(* CODESYS project Johnson,Joachim,Uppgift18_V3.project

Project tree, tasks and I/O mapping:
  Device : CODESYS Control Win V3, 3S - Smart Software Solutions GmbH, order no. 305021, version 3.5.10.40
    application Application
      libraries: Standard, * (System)
      task MainTask (cyclic, interval t#20ms, priority 1) calls PLC_PRG
      program PLC_PRG [LD]
      Symbols
      global variables GVL
*)

// Device/Application/GVL
{attribute 'qualified_only'}
VAR_GLOBAL
		// signals from buttons
	iSUB00_S1: BOOL; // StartButton
	iSUB00_S2: BOOL; // Stopbutton
	iSUB00_S3: BOOL; // Resetbutton
	
	running: BOOL; // Is the aplication running
	alarm: BOOL; // Is the aplication running
	
	// Signals from conveyors
	iSUB01_B1: BOOL; // Signals för conveyor 1. ontop
	iSUB02_B1: BOOL; // Signals för conveyor 2. ontop
	iSUB03_B1: BOOL; // Signals för conveyor 3. ontop
	
	// conveyor signal ontop conveyro.
	oSUB00_H1: BOOL; // Auto-On light
	oSUB00_H2: BOOL; // Alarm light
	oSUB00_H3: WORD;
	oSUB01_K1: BOOL; // MOTOR FÖR converoyr 1
	oSUB02_K1: BOOL; // MOTOR FÖR converoyr 2
	oSUB03_K1: BOOL; // MOTOR FÖR converoyr 3
END_VAR

// Device/Application/PLC_PRG
PROGRAM PLC_PRG
VAR
	ReturnRunnongBool: BOOL;
	PressBtnTime: TIME;
	PressBtnTimer: TON;
	ONTOPCONRETURN: BOOL;
	ONTOPCONRETURN2: BOOL; // check that the previous con not take controll over engine/converour
	ONTOPCONRETURN3: BOOL; // check that the previous con not take controll over engine/converour
	PallCounter: CTU;
END_VAR
VAR // added by the converter: edge detectors and wires of the graphical bodies
    _w1, _w2, _w3, _w4 : BOOL;
END_VAR

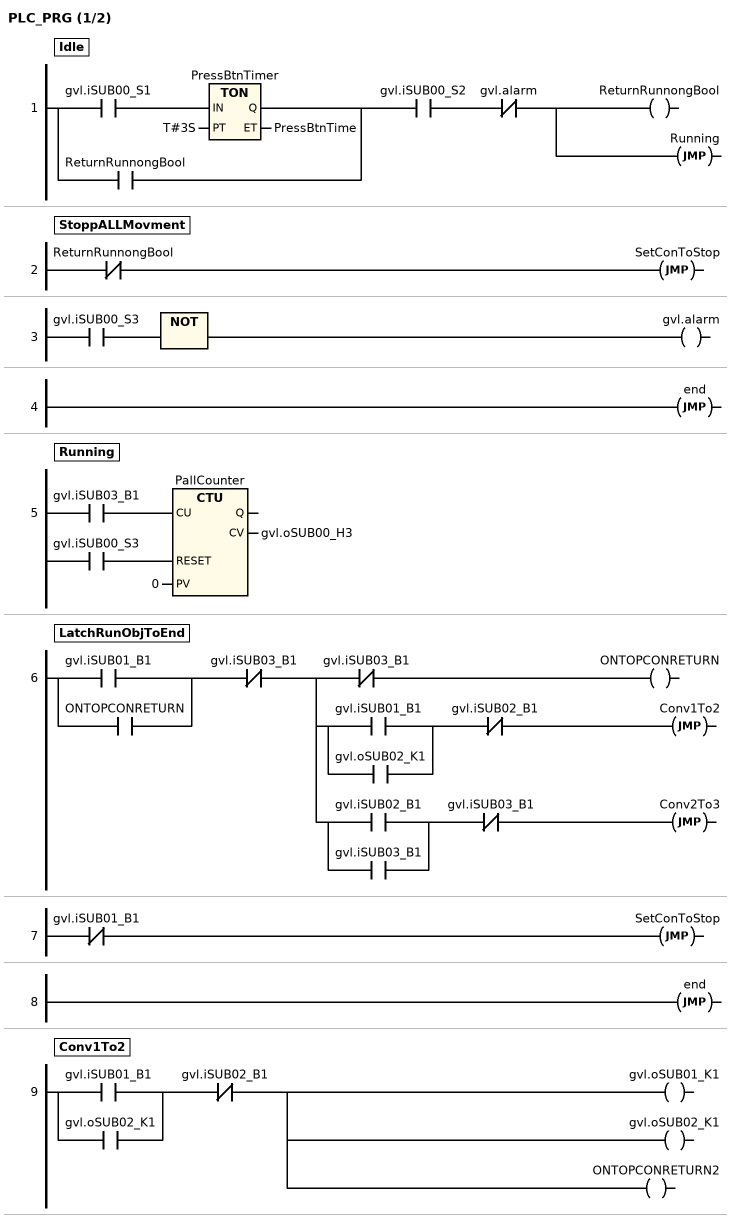
// NETWORK 1
Idle:
PressBtnTimer(IN := gvl.iSUB00_S1, PT := T#3S, ET => PressBtnTime); // TON
_w1 := (PressBtnTimer.Q OR ReturnRunnongBool) AND gvl.iSUB00_S2 AND NOT gvl.alarm;
ReturnRunnongBool := _w1;
IF _w1 THEN JMP Running; END_IF

// NETWORK 2
StoppALLMovment:
IF NOT ReturnRunnongBool THEN JMP SetConToStop; END_IF

// NETWORK 3
gvl.alarm := NOT gvl.iSUB00_S3;

// NETWORK 4
JMP end;

// NETWORK 5
Running:
PallCounter(CU := gvl.iSUB03_B1, RESET := gvl.iSUB00_S3, PV := 0, CV => gvl.oSUB00_H3); // CTU

// NETWORK 6
LatchRunObjToEnd:
_w2 := (gvl.iSUB01_B1 OR ONTOPCONRETURN) AND NOT gvl.iSUB03_B1;
ONTOPCONRETURN := _w2 AND NOT gvl.iSUB03_B1;
IF (_w2 AND (gvl.iSUB01_B1 OR gvl.oSUB02_K1)) AND NOT gvl.iSUB02_B1 THEN JMP Conv1To2; END_IF
IF _w2 AND (gvl.iSUB02_B1 OR gvl.iSUB03_B1) AND NOT gvl.iSUB03_B1 THEN JMP Conv2To3; END_IF

// NETWORK 7
IF NOT gvl.iSUB01_B1 THEN JMP SetConToStop; END_IF

// NETWORK 8
JMP end;

// NETWORK 9
Conv1To2:
_w3 := (gvl.iSUB01_B1 OR gvl.oSUB02_K1) AND NOT gvl.iSUB02_B1;
gvl.oSUB01_K1 := _w3;
gvl.oSUB02_K1 := _w3;
ONTOPCONRETURN2 := _w3;

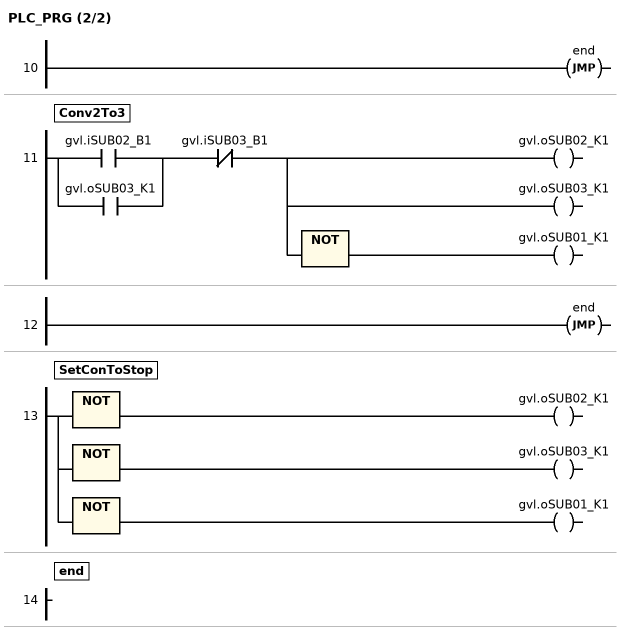
// NETWORK 10
JMP end;

// NETWORK 11
Conv2To3:
_w4 := (gvl.iSUB02_B1 OR gvl.oSUB03_K1) AND NOT gvl.iSUB03_B1;
gvl.oSUB02_K1 := _w4;
gvl.oSUB03_K1 := _w4;
gvl.oSUB01_K1 := NOT _w4;

// NETWORK 12
JMP end;

// NETWORK 13
SetConToStop:
gvl.oSUB02_K1 := NOT TRUE;
gvl.oSUB03_K1 := NOT TRUE;
gvl.oSUB01_K1 := NOT TRUE;

// NETWORK 14
end: ;

END_PROGRAM
